FUNCTION_BLOCK FB_ConvOpen_Check
VAR_INPUT
END_VAR
VAR_OUTPUT
END_VAR
VAR
	
END_VAR

IF IO.bAutoMode THEN
	//receiving status
	IF NOT IO.bConv1_In AND IO.bReCyl1_State_Extend THEN
		IO_Conveyor.bReceiving_State_Open := TRUE ;	
	ELSE
		IO_Conveyor.bReceiving_State_Open := FALSE ;	
	END_IF
	
	//conv1 status
	IF NOT IO.bConv1_Out OR NOT IO.bMotor1 THEN
		IO_Conveyor.bExit1_IsOpen := TRUE ;
	ELSE
		IO_Conveyor.bExit1_IsOpen := FALSE ;
	END_IF	
	
	//conv2 status
	IF NOT IO.bConv2_Out OR NOT IO.bMotor2 THEN
		IO_Conveyor.bExit2_IsOpen := TRUE ;
	ELSE
		IO_Conveyor.bExit2_IsOpen := FALSE ;
	END_IF	
	
	//conv3 status
	IF NOT IO.bConv3_Out OR NOT IO.bMotor3 THEN
		IO_Conveyor.bExit3_IsOpen := TRUE ;
	ELSE
		IO_Conveyor.bExit3_IsOpen := FALSE ;
	END_IF	
	
	//conv4 status
	IF NOT IO.bConv4_Out OR NOT IO.bMotor4 THEN
		IO_Conveyor.bExit4_IsOpen := TRUE ;
	ELSE
		IO_Conveyor.bExit4_IsOpen := FALSE ;
	END_IF
END_IF

END_FUNCTION_BLOCK

(* stored: Version 1.1.0.1, ProductVersion 3.1.4024.12
   POU FB_ConvOpen_Check: Id {0faadb23-fb56-4fe6-be4e-a6dd15fde767}, SpecialFunc None *)
